// TIA Portal V18 export
DATA_BLOCK "ExternalData"   // DB15
{ S7_Optimized_Access := 'FALSE' }
VERSION : 0.1
// stored: AutoNumber true, DBAccessibleFromOPCUA true, DBAccessibleFromWebserver true, IsOnlyStoredInLoadMemory false, IsWriteProtectedInAS false
   VAR
      ex_CoveyorBusy : Array[0..7] of Bool;
      ex_CoveyorSpeed : Array[0..7] of Int;
      ex_CoveyorCount : Array[0..7] of Int;
      ex_RobotSpeed_0 : Int;
      ex_StorerPlaces_0 : Array[0..4] of "udt_StoreRow";
      ex_StorerTypes_0 { S7_SetPoint := 'True'} : Array[0..4] of "udt_StoreRowBoxType";
      ex_status_box_movement : Bool;
      ex_status_robot_movement : Bool;
      ex_status_pallet_movement : Bool;
      ex_status_capacitive_ready : Bool;
      ex_status_storer_movement : Bool;
      ex_beaconGreen : Bool;
      ex_beaconRed : Bool;
      ex_beaconYellow : Bool;
   END_VAR
BEGIN
END_DATA_BLOCK
